TYPE DUT :
STRUCT
END_STRUCT
END_TYPE

(* stored: Version 1.1.0.1, ProductVersion 3.1.4024.12
   DUT DUT: Id {885704cf-2793-47f7-904f-10a1384dfaca} *)
